{attribute 'qualified_only'}
{attribute 'strict'}
TYPE E_FaultLevel :
(
	DIAGNOSTIC 		:= 0,
	LOW 			:= 1,
	MEDIUM			:= 2,
	HIGH			:= 3,
	CRITICAL		:= 4
);
END_TYPE

(* stored: Version 1.1.0.1, ProductVersion 3.1.4024.13
   EnumerationTextList E_FaultLevel: Id {09ed1a9d-c7e3-46c7-b801-145016d9b09d} *)
